TYPE Kraftvariablen :
STRUCT
	Fx					:LREAL;							// Kraft in X-Richtung 
	Fy					:LREAL;							// Kraft in Y-Richtung 
	Fz					:LREAL;							// Kraft in Z-Richtung 
	Tx					:LREAL;							// Moment auf X-Achse 
	Ty					:LREAL;							// Moment auf Y-Achse 
	Tz					:LREAL;							// Moment auf Z-Achse 
END_STRUCT
END_TYPE

(* stored: Version 1.1.0.1
   DUT Kraftvariablen: Id {02ad4d97-762c-47de-a2f1-7a6877800f4b} *)
